FUNCTION_BLOCK SK_Dwell (* Skill primitive Dwell: Wait at the current position (stands in for dispensing until there is a pump) (parameters: Duration [s] 0.0..60.0, default 1.0). OPC UA Start(Session, parameters...)/Stop/Abort/Reset(Session) -> [Accepted, ErrorID]; START/HALT/ABORT/RESET from a parent -> SUCCESS or FAILURE(ErrorID) *)
  (* Standard: 61499-2 *)
  (* Version 0.1, 2026-09-28, Project contributors, AAU Smart Production Lab *)
  PACKAGE filling;
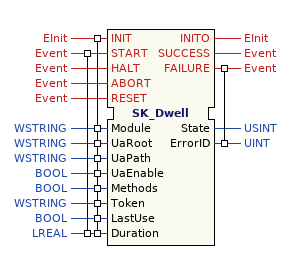
  EVENT_INPUT
    INIT : EInit WITH Module, UaRoot, UaPath, UaEnable, Methods, Token, LastUse, Duration;
    START WITH Duration;
    HALT;
    ABORT;
    RESET;
  END_EVENT
  EVENT_OUTPUT
    INITO : EInit;
    SUCCESS;
    FAILURE WITH ErrorID;
  END_EVENT
  VAR_INPUT
    Module : WSTRING;
    UaRoot : WSTRING;
    UaPath : WSTRING;
    UaEnable : BOOL;
    Methods : BOOL;
    Token : WSTRING;
    LastUse : BOOL := TRUE;
    Duration : LREAL := 1.0;
  END_VAR
  VAR_OUTPUT
    State : USINT;
    ErrorID : UINT;
  END_VAR
  (* Group SkillControl: State machine and OPC UA: Start(Session, parameters) with the range check, Stop, Abort, Reset; State, parameters and results published *)
  (* Group Execution: One run: the contract, the command to the equipment and the end condition *)
  FBS
    Control : modlib::SKILL_Core; {SET_ATTRIBUTE(GroupName, SkillControl)}
    Logic : filling::SL_Dwell; {SET_ATTRIBUTE(GroupName, Execution)}
    UaStart : iec61499::net::SERVER_2_2; {SET_ATTRIBUTE(GroupName, SkillControl)}
    Par_Duration : modlib::SKILL_Param_LREAL(Lower := 0.0, Upper := 60.0); {SET_ATTRIBUTE(GroupName, SkillControl)}
    PubParams : iec61499::net::PUBLISH_1; {SET_ATTRIBUTE(GroupName, SkillControl)}
    Timer : iec61499::events::E_DELAY; {SET_ATTRIBUTE(GroupName, Execution)}
  END_FBS
  EVENT_CONNECTIONS
    Control.RSP_START TO UaStart.RSP;
    UaStart.IND TO Par_Duration.CHECK;
    Control.GO TO Par_Duration.LATCH;
    Par_Duration.CHECKED TO Control.CMD_START;
    Par_Duration.LATCHED TO PubParams.REQ;
    PubParams.INITO TO PubParams.REQ;
    INIT TO Control.INIT;
    Control.INITO TO Logic.INIT;
    Logic.INITO TO UaStart.INIT;
    UaStart.INITO TO Par_Duration.INIT;
    Par_Duration.INITO TO PubParams.INIT;
    PubParams.INITO TO INITO;
    START TO Control.START;
    HALT TO Control.HALT;
    ABORT TO Control.ABORT;
    RESET TO Control.RESET;
    Control.SUCCESS TO SUCCESS;
    Control.FAILURE TO FAILURE;
    Par_Duration.LATCHED TO Logic.START;
    Control.HALT_O TO Logic.HALT;
    Control.ABORT_O TO Logic.ABORT;
    Control.RUN_STOP TO Control.STOP_DONE;
    Logic.DONE TO Control.EXEC_DONE;
    Logic.FAILED TO Control.EXEC_FAILED;
    Logic.HALTED TO Control.EXEC_FAILED;
    Logic.TIMER_START TO Timer.START;
    Logic.TIMER_STOP TO Timer.STOP;
    Timer.EO TO Logic.TIMER;
  END_CONNECTIONS
  DATA_CONNECTIONS
    Control.IdStart TO UaStart.ID;
    UaStart.RD_1 TO Control.S_Start;
    Control.Accepted TO UaStart.SD_1;
    Control.RspError TO UaStart.SD_2;
    UaStart.RD_2 TO Par_Duration.S;
    Control.FromUa TO Par_Duration.FromUa;
    Par_Duration.P TO PubParams.SD_1;
    Par_Duration.InRange TO Control.InRange;
    Module TO Control.Module;
    UaRoot TO Control.UaRoot;
    UaPath TO Control.UaPath;
    UaEnable TO Control.UaEnable;
    Methods TO Control.Methods;
    Methods TO UaStart.QI;
    Control.State TO State;
    Control.ErrorID TO ErrorID;
    UaRoot TO Logic.UaRoot;
    UaPath TO Logic.UaPath;
    UaEnable TO PubParams.QI;
    Logic.IdParams TO PubParams.ID;
    Duration TO Par_Duration.Default;
    Par_Duration.P TO Logic.Duration;
    Logic.ErrorID TO Control.ExecError;
    Logic.TimerDT TO Timer.DT;
  END_CONNECTIONS
END_FUNCTION_BLOCK
